(* PLC project SmartTextile_Ladder, Eesha Masand Smart Textile Manufacturing 2 *)
(* stored: creationDateTime 2026-10-07T12:00:00, modificationDateTime 2026-10-07T12:00:00 *)

(* Smart textile line: control logic as a ladder diagram. Runs first in the scan. *)
PROGRAM SmartTextileLadder
  VAR
    X0_StartPB AT %QX102.0 : BOOL;  (* X0: Start push-button (physical) *)
    X1_StopPB AT %QX102.1 : BOOL;  (* X1: Stop push-button (physical) *)
    X2_ResetPB AT %QX102.2 : BOOL;  (* X2: Reset push-button (physical) *)
    X3_AtS1_FeedId AT %QX102.3 : BOOL;  (* X3: Product at station 1: feed / identification *)
    X4_TypeA_Sensor AT %QX102.4 : BOOL;  (* X4: Type A sensor *)
    X5_TypeB_Sensor AT %QX102.5 : BOOL;  (* X5: Type B sensor *)
    X6_AtS2_Cutting AT %QX102.6 : BOOL;  (* X6: Product at station 2: cutting *)
    X7_AtS3_Finishing AT %QX102.7 : BOOL;  (* X7: Product at station 3: finishing *)
    X10_AtS4_Inspection AT %QX103.0 : BOOL;  (* X10: Product at station 4: inspection *)
    X11_InspComplete AT %QX103.1 : BOOL;  (* X11: Inspection complete (vision result valid) *)
    X12_DefectDetected AT %QX103.2 : BOOL;  (* X12: Defect detected by vision *)
    X13_RobotReady AT %QX103.3 : BOOL;  (* X13: Robot ready (home position) *)
    X14_RobotPlaceDone AT %QX103.4 : BOOL;  (* X14: Robot place done *)
    X15_PackComplete AT %QX103.5 : BOOL;  (* X15: Packaging complete *)
    X16_RobotHealthy AT %QX103.6 : BOOL;  (* X16: Robot healthy (NC wiring: ON = OK, OFF = fault) *)
    X17_EStopOK AT %QX103.7 : BOOL;  (* X17: Emergency stop chain (NC wiring: ON = released, OFF = pressed) *)
    X20_AtS5_Robot AT %QX104.0 : BOOL;  (* X20: Product at station 5: robot pick *)
    Y0_FeederMotor AT %QX0.0 : BOOL;  (* Y0: Feeder motor *)
    Y1_MainConveyor AT %QX0.1 : BOOL;  (* Y1: Main conveyor *)
    Y2_Cutter AT %QX0.2 : BOOL;  (* Y2: Cutter (stage 1) *)
    Y3_HeatPress AT %QX0.3 : BOOL;  (* Y3: Heat press (stage 2) *)
    Y4_InspTrigger AT %QX0.4 : BOOL;  (* Y4: Inspection trigger (camera) *)
    Y5_RobotPickReq AT %QX0.5 : BOOL;  (* Y5: Robot pick request *)
    Y6_DestGood AT %QX0.6 : BOOL;  (* Y6: Robot destination: good *)
    Y7_DestReject AT %QX0.7 : BOOL;  (* Y7: Robot destination: reject *)
    Y10_PackMachine AT %QX1.0 : BOOL;  (* Y10: Packaging machine *)
    Y11_AlarmBuzzer AT %QX1.1 : BOOL;  (* Y11: Alarm buzzer *)
    Y12_RunLamp AT %QX1.2 : BOOL;  (* Y12: Run lamp (green) *)
    Y13_FaultLamp AT %QX1.3 : BOOL;  (* Y13: Fault / E-stop lamp (red) *)
    M100_HmiStart AT %QX100.0 : BOOL;  (* M100: HMI start button *)
    M101_HmiStop AT %QX100.1 : BOOL;  (* M101: HMI stop button *)
    M102_HmiReset AT %QX100.2 : BOOL;  (* M102: HMI reset button *)
    M103_HmiAuto AT %QX100.3 : BOOL;  (* M103: HMI auto mode button *)
    M104_HmiManual AT %QX100.4 : BOOL;  (* M104: HMI manual mode button *)
    M105_HmiProdA AT %QX100.5 : BOOL;  (* M105: HMI product A override *)
    M106_HmiProdB AT %QX100.6 : BOOL;  (* M106: HMI product B override *)
    M107_HmiClear AT %QX100.7 : BOOL;  (* M107: HMI clear counters button *)
    M108_HmiEStop AT %QX101.0 : BOOL;  (* M108: HMI emergency stop button *)
    M0_SystemRun AT %QX105.0 : BOOL;  (* M0: System run *)
    M1_Fault AT %QX105.1 : BOOL;  (* M1: Fault latched *)
    M2_EStop AT %QX105.2 : BOOL;  (* M2: Emergency stop latched *)
    M31_ManualMode AT %QX105.3 : BOOL;  (* M31: Manual mode (0 = auto) *)
    M17_ManualTypeB AT %QX105.4 : BOOL;  (* M17: Manual product selection (0 = A, 1 = B) *)
    M3_PhaseIndex AT %QX105.5 : BOOL;  (* M3: Phase: conveyor indexing *)
    M4_PhaseWork AT %QX105.6 : BOOL;  (* M4: Phase: stations working *)
    M75_PackBusy AT %QX105.7 : BOOL;  (* M75: Packaging machine busy *)
    M50_S1_Occupied AT %QX106.0 : BOOL;  (* M50: Station 1 occupied *)
    M51_S2_Occupied AT %QX106.1 : BOOL;  (* M51: Station 2 occupied *)
    M52_S3_Occupied AT %QX106.2 : BOOL;  (* M52: Station 3 occupied *)
    M53_S4_Occupied AT %QX106.3 : BOOL;  (* M53: Station 4 occupied *)
    M54_S5_Occupied AT %QX106.4 : BOOL;  (* M54: Station 5 occupied *)
    M55_DefectAtS4 AT %QX106.5 : BOOL;  (* M55: Defect flag of the product at station 4 *)
    M56_DefectAtS5 AT %QX106.6 : BOOL;  (* M56: Defect flag of the product at station 5 *)
    M60_S1_IsTypeB AT %QX107.0 : BOOL;  (* M60: Product at station 1 is type B *)
    M61_S2_IsTypeB AT %QX107.1 : BOOL;  (* M61: Product at station 2 is type B *)
    M62_S3_IsTypeB AT %QX107.2 : BOOL;  (* M62: Product at station 3 is type B *)
    M63_S4_IsTypeB AT %QX107.3 : BOOL;  (* M63: Product at station 4 is type B *)
    M64_S5_IsTypeB AT %QX107.4 : BOOL;  (* M64: Product at station 5 is type B *)
  END_VAR
  VAR
    M69_FeedDone : BOOL;  (* M69: Feed time elapsed in this work phase *)
    M70_S1_IdDone : BOOL;  (* M70: Station 1 identification done *)
    M71_S2_CutDone : BOOL;  (* M71: Station 2 cutting done *)
    M72_S3_FinishDone : BOOL;  (* M72: Station 3 finishing done *)
    M73_S4_InspDone : BOOL;  (* M73: Station 4 inspection result latched *)
    M80_S1_Departed : BOOL;  (* M80: Old product has left station 1 (this index) *)
    M81_S2_Departed : BOOL;  (* M81: Old product has left station 2 (this index) *)
    M82_S3_Departed : BOOL;  (* M82: Old product has left station 3 (this index) *)
    M83_S4_Departed : BOOL;  (* M83: Old product has left station 4 (this index) *)
    M84_S5_Departed : BOOL;  (* M84: Old product has left station 5 (this index) *)
    M22_GoodSorted : BOOL;  (* M22: Good product sorted (pulse) *)
    M23_RejectSorted : BOOL;  (* M23: Reject product sorted (pulse) *)
    M24_IndexComplete : BOOL;  (* M24: Index complete: all products at next station *)
    M25_WorkComplete : BOOL;  (* M25: Work complete: all stations finished *)
    M26_StationsDone : BOOL;  (* M26: All occupied stations finished their task *)
    M28_AllDeparted : BOOL;  (* M28: Every old product has left its station *)
    M29_AllArrived : BOOL;  (* M29: Every expected product reached its station *)
    M32_PackagedPulse : BOOL;  (* M32: Product packaged (pulse) *)
  END_VAR
  VAR_EXTERNAL
    T0_FeedTime_Q : BOOL;  (* Shared with the data program *)
    T1_CutTime_Q : BOOL;  (* Shared with the data program *)
    T2_FinishA_Q : BOOL;  (* Shared with the data program *)
    T3_FinishB_Q : BOOL;  (* Shared with the data program *)
    T4_InspTimeout_Q : BOOL;  (* Shared with the data program *)
    T7_IndexWdg_Q : BOOL;  (* Shared with the data program *)
    T8_IdDwell_Q : BOOL;  (* Shared with the data program *)
    T9_IdTimeout_Q : BOOL;  (* Shared with the data program *)
    T10_RobotWdg_Q : BOOL;  (* Shared with the data program *)
    T11_PackWdg_Q : BOOL;  (* Shared with the data program *)
    F_R01_RobotFaultRobot : BOOL;  (* Shared with the data program *)
    F_R02_InspectionTimeoutVision : BOOL;  (* Shared with the data program *)
    F_R03_IndexPackagingTimeout : BOOL;  (* Shared with the data program *)
    F_R04_UnknownProductIdentification : BOOL;  (* Shared with the data program *)
    F_R05_EmergencyStopChain : BOOL;  (* Shared with the data program *)
    F_R06_ResetClearFaults : BOOL;  (* Shared with the data program *)
    F_R11_ManualOverrideProduct : BOOL;  (* Shared with the data program *)
    F_R12_ManualOverrideProduct : BOOL;  (* Shared with the data program *)
    F_R13_IdleStartFeed : BOOL;  (* Shared with the data program *)
    F_R26_IndexWork : BOOL;  (* Shared with the data program *)
    F_R27_FeederStartBelt : BOOL;  (* Shared with the data program *)
    F_R29_IdentificationDwell : BOOL;  (* Shared with the data program *)
    F_R30_IdentificationTimeout : BOOL;  (* Shared with the data program *)
    F_R31_IdentifyProductAuto : BOOL;  (* Shared with the data program *)
    F_R32_IdentifyProductB : BOOL;  (* Shared with the data program *)
    F_R35_CutterCuttingTime : BOOL;  (* Shared with the data program *)
    F_R38_FinishingTimeProduct : BOOL;  (* Shared with the data program *)
    F_R39_FinishingTimeProduct : BOOL;  (* Shared with the data program *)
    F_R42_InspectionTimeoutTimer : BOOL;  (* Shared with the data program *)
    F_R49_RobotWatchdogTimer : BOOL;  (* Shared with the data program *)
    F_R54_PackagingMachineWatchdog : BOOL;  (* Shared with the data program *)
    F_R59_WorkIndex : BOOL;  (* Shared with the data program *)
    F_R61_IndexWatchdog15 : BOOL;  (* Shared with the data program *)
    F_R62_StopwatchesAddOne : BOOL;  (* Shared with the data program *)
    F_R63_TaktTimeLast : BOOL;  (* Shared with the data program *)
    F_R64_GoodCounter : BOOL;  (* Shared with the data program *)
    F_R65_RejectCounter : BOOL;  (* Shared with the data program *)
    F_R66_PackagedCounter : BOOL;  (* Shared with the data program *)
    F_R71_ClearCountersKPIs : BOOL;  (* Shared with the data program *)
  END_VAR
  VAR  (* added by the conversion: wires and edge detectors of the diagram *)
    R_TRIG1 : R_TRIG;
    R_TRIG2 : R_TRIG;
    R_TRIG3 : R_TRIG;
    R_TRIG4 : R_TRIG;
    R_TRIG5 : R_TRIG;
    R_TRIG6 : R_TRIG;
    R_TRIG7 : R_TRIG;
    R_TRIG8 : R_TRIG;
  END_VAR

(* LD diagram, written out as Structured Text *)
IF NOT X16_RobotHealthy OR T10_RobotWdg_Q THEN M1_Fault := TRUE; END_IF;
F_R01_RobotFaultRobot := NOT X16_RobotHealthy OR T10_RobotWdg_Q;
IF T4_InspTimeout_Q THEN M1_Fault := TRUE; END_IF;
F_R02_InspectionTimeoutVision := T4_InspTimeout_Q;
IF T7_IndexWdg_Q OR T11_PackWdg_Q THEN M1_Fault := TRUE; END_IF;
F_R03_IndexPackagingTimeout := T7_IndexWdg_Q OR T11_PackWdg_Q;
IF T9_IdTimeout_Q THEN M1_Fault := TRUE; END_IF;
F_R04_UnknownProductIdentification := T9_IdTimeout_Q;
R_TRIG1(CLK := M108_HmiEStop);
F_R05_EmergencyStopChain := NOT X17_EStopOK OR R_TRIG1.Q OR M2_EStop;
IF F_R05_EmergencyStopChain THEN M2_EStop := TRUE; END_IF;
R_TRIG2(CLK := M102_HmiReset);
R_TRIG3(CLK := X2_ResetPB);
F_R06_ResetClearFaults := (R_TRIG2.Q OR R_TRIG3.Q) AND X16_RobotHealthy AND X17_EStopOK;
IF F_R06_ResetClearFaults THEN M1_Fault := FALSE; END_IF;
IF F_R06_ResetClearFaults THEN M2_EStop := FALSE; END_IF;
IF F_R06_ResetClearFaults THEN M3_PhaseIndex := FALSE; END_IF;
IF F_R06_ResetClearFaults THEN M4_PhaseWork := FALSE; END_IF;
IF F_R06_ResetClearFaults THEN M50_S1_Occupied := FALSE; END_IF;
IF F_R06_ResetClearFaults THEN M51_S2_Occupied := FALSE; END_IF;
IF F_R06_ResetClearFaults THEN M52_S3_Occupied := FALSE; END_IF;
IF F_R06_ResetClearFaults THEN M53_S4_Occupied := FALSE; END_IF;
IF F_R06_ResetClearFaults THEN M54_S5_Occupied := FALSE; END_IF;
IF F_R06_ResetClearFaults THEN M55_DefectAtS4 := FALSE; END_IF;
IF F_R06_ResetClearFaults THEN M56_DefectAtS5 := FALSE; END_IF;
IF F_R06_ResetClearFaults THEN M60_S1_IsTypeB := FALSE; END_IF;
IF F_R06_ResetClearFaults THEN M61_S2_IsTypeB := FALSE; END_IF;
IF F_R06_ResetClearFaults THEN M62_S3_IsTypeB := FALSE; END_IF;
IF F_R06_ResetClearFaults THEN M63_S4_IsTypeB := FALSE; END_IF;
IF F_R06_ResetClearFaults THEN M64_S5_IsTypeB := FALSE; END_IF;
IF F_R06_ResetClearFaults THEN M69_FeedDone := FALSE; END_IF;
IF F_R06_ResetClearFaults THEN M70_S1_IdDone := FALSE; END_IF;
IF F_R06_ResetClearFaults THEN M71_S2_CutDone := FALSE; END_IF;
IF F_R06_ResetClearFaults THEN M72_S3_FinishDone := FALSE; END_IF;
IF F_R06_ResetClearFaults THEN M73_S4_InspDone := FALSE; END_IF;
IF F_R06_ResetClearFaults THEN M75_PackBusy := FALSE; END_IF;
IF F_R06_ResetClearFaults THEN M80_S1_Departed := FALSE; END_IF;
IF F_R06_ResetClearFaults THEN M81_S2_Departed := FALSE; END_IF;
IF F_R06_ResetClearFaults THEN M82_S3_Departed := FALSE; END_IF;
IF F_R06_ResetClearFaults THEN M83_S4_Departed := FALSE; END_IF;
IF F_R06_ResetClearFaults THEN M84_S5_Departed := FALSE; END_IF;
R_TRIG4(CLK := M100_HmiStart);
R_TRIG5(CLK := X0_StartPB);
IF (R_TRIG4.Q OR R_TRIG5.Q) AND NOT M1_Fault AND NOT M2_EStop AND X16_RobotHealthy AND X17_EStopOK THEN M0_SystemRun := TRUE; END_IF;
IF M101_HmiStop OR X1_StopPB OR NOT X16_RobotHealthy OR NOT X17_EStopOK OR M1_Fault OR M2_EStop THEN M0_SystemRun := FALSE; END_IF;
IF M103_HmiAuto THEN M31_ManualMode := FALSE; END_IF;
IF M104_HmiManual THEN M31_ManualMode := TRUE; END_IF;
IF M105_HmiProdA AND M31_ManualMode THEN M17_ManualTypeB := FALSE; END_IF;
F_R11_ManualOverrideProduct := M105_HmiProdA AND M31_ManualMode;
IF M106_HmiProdB AND M31_ManualMode THEN M17_ManualTypeB := TRUE; END_IF;
F_R12_ManualOverrideProduct := M106_HmiProdB AND M31_ManualMode;
F_R13_IdleStartFeed := M0_SystemRun AND NOT M3_PhaseIndex AND NOT M4_PhaseWork AND NOT M1_Fault AND NOT M2_EStop;
IF F_R13_IdleStartFeed THEN M4_PhaseWork := TRUE; END_IF;
M28_AllDeparted := M0_SystemRun AND M3_PhaseIndex AND (NOT M50_S1_Occupied OR M80_S1_Departed) AND (NOT M51_S2_Occupied OR M81_S2_Departed) AND (NOT M52_S3_Occupied OR M82_S3_Departed) AND (NOT M53_S4_Occupied OR M83_S4_Departed) AND (NOT M54_S5_Occupied OR M84_S5_Departed);
M29_AllArrived := M0_SystemRun AND M3_PhaseIndex AND X3_AtS1_FeedId AND (NOT M50_S1_Occupied OR X6_AtS2_Cutting) AND (NOT M51_S2_Occupied OR X7_AtS3_Finishing) AND (NOT M52_S3_Occupied OR X10_AtS4_Inspection) AND (NOT M53_S4_Occupied OR X20_AtS5_Robot);
M24_IndexComplete := M28_AllDeparted AND M29_AllArrived;
IF M0_SystemRun AND M3_PhaseIndex AND M50_S1_Occupied AND NOT X3_AtS1_FeedId THEN M80_S1_Departed := TRUE; END_IF;
IF M0_SystemRun AND M3_PhaseIndex AND M51_S2_Occupied AND NOT X6_AtS2_Cutting THEN M81_S2_Departed := TRUE; END_IF;
IF M0_SystemRun AND M3_PhaseIndex AND M52_S3_Occupied AND NOT X7_AtS3_Finishing THEN M82_S3_Departed := TRUE; END_IF;
IF M0_SystemRun AND M3_PhaseIndex AND M53_S4_Occupied AND NOT X10_AtS4_Inspection THEN M83_S4_Departed := TRUE; END_IF;
IF M0_SystemRun AND M3_PhaseIndex AND M54_S5_Occupied AND NOT X20_AtS5_Robot THEN M84_S5_Departed := TRUE; END_IF;
IF M24_IndexComplete AND M53_S4_Occupied THEN M54_S5_Occupied := TRUE; END_IF;
IF M24_IndexComplete AND NOT M53_S4_Occupied THEN M54_S5_Occupied := FALSE; END_IF;
IF M24_IndexComplete AND M52_S3_Occupied THEN M53_S4_Occupied := TRUE; END_IF;
IF M24_IndexComplete AND NOT M52_S3_Occupied THEN M53_S4_Occupied := FALSE; END_IF;
IF M24_IndexComplete AND M51_S2_Occupied THEN M52_S3_Occupied := TRUE; END_IF;
IF M24_IndexComplete AND NOT M51_S2_Occupied THEN M52_S3_Occupied := FALSE; END_IF;
IF M24_IndexComplete AND M50_S1_Occupied THEN M51_S2_Occupied := TRUE; END_IF;
IF M24_IndexComplete AND NOT M50_S1_Occupied THEN M51_S2_Occupied := FALSE; END_IF;
IF M24_IndexComplete THEN M50_S1_Occupied := TRUE; END_IF;
IF M24_IndexComplete AND M63_S4_IsTypeB THEN M64_S5_IsTypeB := TRUE; END_IF;
IF M24_IndexComplete AND NOT M63_S4_IsTypeB THEN M64_S5_IsTypeB := FALSE; END_IF;
IF M24_IndexComplete AND M62_S3_IsTypeB THEN M63_S4_IsTypeB := TRUE; END_IF;
IF M24_IndexComplete AND NOT M62_S3_IsTypeB THEN M63_S4_IsTypeB := FALSE; END_IF;
IF M24_IndexComplete AND M61_S2_IsTypeB THEN M62_S3_IsTypeB := TRUE; END_IF;
IF M24_IndexComplete AND NOT M61_S2_IsTypeB THEN M62_S3_IsTypeB := FALSE; END_IF;
IF M24_IndexComplete AND M60_S1_IsTypeB THEN M61_S2_IsTypeB := TRUE; END_IF;
IF M24_IndexComplete AND NOT M60_S1_IsTypeB THEN M61_S2_IsTypeB := FALSE; END_IF;
IF M24_IndexComplete THEN M60_S1_IsTypeB := FALSE; END_IF;
IF M24_IndexComplete AND M55_DefectAtS4 THEN M56_DefectAtS5 := TRUE; END_IF;
IF M24_IndexComplete AND NOT M55_DefectAtS4 THEN M56_DefectAtS5 := FALSE; END_IF;
IF M24_IndexComplete THEN M55_DefectAtS4 := FALSE; END_IF;
IF M24_IndexComplete THEN M69_FeedDone := FALSE; END_IF;
IF M24_IndexComplete THEN M70_S1_IdDone := FALSE; END_IF;
IF M24_IndexComplete THEN M71_S2_CutDone := FALSE; END_IF;
IF M24_IndexComplete THEN M72_S3_FinishDone := FALSE; END_IF;
IF M24_IndexComplete THEN M73_S4_InspDone := FALSE; END_IF;
IF M24_IndexComplete THEN M80_S1_Departed := FALSE; END_IF;
IF M24_IndexComplete THEN M81_S2_Departed := FALSE; END_IF;
IF M24_IndexComplete THEN M82_S3_Departed := FALSE; END_IF;
IF M24_IndexComplete THEN M83_S4_Departed := FALSE; END_IF;
IF M24_IndexComplete THEN M84_S5_Departed := FALSE; END_IF;
IF M24_IndexComplete THEN M3_PhaseIndex := FALSE; END_IF;
IF M24_IndexComplete THEN M4_PhaseWork := TRUE; END_IF;
F_R26_IndexWork := M24_IndexComplete;
Y0_FeederMotor := M0_SystemRun AND M4_PhaseWork AND NOT M69_FeedDone;
F_R27_FeederStartBelt := M0_SystemRun AND M4_PhaseWork AND NOT M69_FeedDone;
IF T0_FeedTime_Q THEN M69_FeedDone := TRUE; END_IF;
F_R29_IdentificationDwell := M0_SystemRun AND M4_PhaseWork AND M50_S1_Occupied AND X3_AtS1_FeedId;
F_R30_IdentificationTimeout := M0_SystemRun AND M4_PhaseWork AND M50_S1_Occupied AND X3_AtS1_FeedId AND NOT M70_S1_IdDone;
IF T8_IdDwell_Q AND NOT M31_ManualMode AND X4_TypeA_Sensor AND NOT X5_TypeB_Sensor THEN M60_S1_IsTypeB := FALSE; END_IF;
F_R31_IdentifyProductAuto := T8_IdDwell_Q AND NOT M31_ManualMode AND X4_TypeA_Sensor AND NOT X5_TypeB_Sensor;
IF T8_IdDwell_Q AND NOT M31_ManualMode AND X5_TypeB_Sensor AND NOT X4_TypeA_Sensor THEN M60_S1_IsTypeB := TRUE; END_IF;
F_R32_IdentifyProductB := T8_IdDwell_Q AND NOT M31_ManualMode AND X5_TypeB_Sensor AND NOT X4_TypeA_Sensor;
IF T8_IdDwell_Q AND M31_ManualMode AND M17_ManualTypeB THEN M60_S1_IsTypeB := TRUE; END_IF;
IF T8_IdDwell_Q AND M31_ManualMode AND NOT M17_ManualTypeB THEN M60_S1_IsTypeB := FALSE; END_IF;
IF T8_IdDwell_Q AND (M31_ManualMode OR X4_TypeA_Sensor AND NOT X5_TypeB_Sensor OR NOT X4_TypeA_Sensor AND X5_TypeB_Sensor) THEN M70_S1_IdDone := TRUE; END_IF;
Y2_Cutter := M0_SystemRun AND M4_PhaseWork AND M51_S2_Occupied AND X6_AtS2_Cutting AND NOT M71_S2_CutDone;
F_R35_CutterCuttingTime := M0_SystemRun AND M4_PhaseWork AND M51_S2_Occupied AND X6_AtS2_Cutting AND NOT M71_S2_CutDone;
IF T1_CutTime_Q THEN M71_S2_CutDone := TRUE; END_IF;
Y3_HeatPress := M0_SystemRun AND M4_PhaseWork AND M52_S3_Occupied AND X7_AtS3_Finishing AND NOT M72_S3_FinishDone;
F_R38_FinishingTimeProduct := M0_SystemRun AND M4_PhaseWork AND M52_S3_Occupied AND X7_AtS3_Finishing AND NOT M72_S3_FinishDone AND NOT M62_S3_IsTypeB;
F_R39_FinishingTimeProduct := M0_SystemRun AND M4_PhaseWork AND M52_S3_Occupied AND X7_AtS3_Finishing AND NOT M72_S3_FinishDone AND M62_S3_IsTypeB;
IF T2_FinishA_Q OR T3_FinishB_Q THEN M72_S3_FinishDone := TRUE; END_IF;
Y4_InspTrigger := M0_SystemRun AND M4_PhaseWork AND M53_S4_Occupied AND X10_AtS4_Inspection AND NOT M73_S4_InspDone;
F_R42_InspectionTimeoutTimer := M0_SystemRun AND M4_PhaseWork AND M53_S4_Occupied AND X10_AtS4_Inspection AND NOT M73_S4_InspDone AND NOT X11_InspComplete;
IF M0_SystemRun AND M4_PhaseWork AND M53_S4_Occupied AND X10_AtS4_Inspection AND X11_InspComplete AND NOT X12_DefectDetected THEN M55_DefectAtS4 := FALSE; END_IF;
IF M0_SystemRun AND M4_PhaseWork AND M53_S4_Occupied AND X10_AtS4_Inspection AND X11_InspComplete AND X12_DefectDetected THEN M55_DefectAtS4 := TRUE; END_IF;
IF M0_SystemRun AND M4_PhaseWork AND M53_S4_Occupied AND X10_AtS4_Inspection AND X11_InspComplete THEN M73_S4_InspDone := TRUE; END_IF;
Y5_RobotPickReq := M0_SystemRun AND M4_PhaseWork AND M54_S5_Occupied AND X20_AtS5_Robot AND NOT X14_RobotPlaceDone AND (M56_DefectAtS5 OR NOT M75_PackBusy);
Y6_DestGood := M0_SystemRun AND M4_PhaseWork AND M54_S5_Occupied AND NOT M56_DefectAtS5;
Y7_DestReject := M0_SystemRun AND M4_PhaseWork AND M54_S5_Occupied AND M56_DefectAtS5;
F_R49_RobotWatchdogTimer := M0_SystemRun AND M4_PhaseWork AND M54_S5_Occupied;
R_TRIG6(CLK := X14_RobotPlaceDone);
M22_GoodSorted := M0_SystemRun AND M4_PhaseWork AND M54_S5_Occupied AND NOT M56_DefectAtS5 AND R_TRIG6.Q;
R_TRIG7(CLK := X14_RobotPlaceDone);
M23_RejectSorted := M0_SystemRun AND M4_PhaseWork AND M54_S5_Occupied AND M56_DefectAtS5 AND R_TRIG7.Q;
IF M22_GoodSorted OR M23_RejectSorted THEN M54_S5_Occupied := FALSE; END_IF;
IF M22_GoodSorted THEN M75_PackBusy := TRUE; END_IF;
Y10_PackMachine := M0_SystemRun AND M75_PackBusy;
F_R54_PackagingMachineWatchdog := M0_SystemRun AND M75_PackBusy;
R_TRIG8(CLK := X15_PackComplete);
M32_PackagedPulse := M0_SystemRun AND M75_PackBusy AND R_TRIG8.Q;
IF M32_PackagedPulse THEN M75_PackBusy := FALSE; END_IF;
M26_StationsDone := (NOT M50_S1_Occupied OR M70_S1_IdDone) AND (NOT M51_S2_Occupied OR M71_S2_CutDone) AND (NOT M52_S3_Occupied OR M72_S3_FinishDone) AND (NOT M53_S4_Occupied OR M73_S4_InspDone) AND NOT M54_S5_Occupied;
M25_WorkComplete := M0_SystemRun AND M4_PhaseWork AND M69_FeedDone AND M26_StationsDone AND X13_RobotReady;
IF M25_WorkComplete THEN M4_PhaseWork := FALSE; END_IF;
IF M25_WorkComplete THEN M3_PhaseIndex := TRUE; END_IF;
F_R59_WorkIndex := M25_WorkComplete;
Y1_MainConveyor := M0_SystemRun AND M3_PhaseIndex AND NOT M24_IndexComplete;
F_R61_IndexWatchdog15 := M0_SystemRun AND M3_PhaseIndex;
F_R62_StopwatchesAddOne := M0_SystemRun AND (M3_PhaseIndex OR M4_PhaseWork);
F_R63_TaktTimeLast := M22_GoodSorted OR M23_RejectSorted;
F_R64_GoodCounter := M22_GoodSorted;
F_R65_RejectCounter := M23_RejectSorted;
F_R66_PackagedCounter := M32_PackagedPulse;
F_R71_ClearCountersKPIs := M107_HmiClear;
Y12_RunLamp := M0_SystemRun;
Y11_AlarmBuzzer := M1_Fault OR M2_EStop;
Y13_FaultLamp := M1_Fault OR M2_EStop;
END_PROGRAM

(* Timers, counters, fault code, phase and KPI maths. Runs second in the scan. *)
PROGRAM SmartTextileData
  VAR
    D100_GoodCount AT %MW0 : INT;  (* D100: Good count *)
    D101_RejectCount AT %MW1 : INT;  (* D101: Reject count *)
    D102_TotalCount AT %MW2 : INT;  (* D102: Total count *)
    D103_DefectPctX100 AT %MW3 : INT;  (* D103: Defect percentage x100 (1670 = 16.70 %) *)
    D104_TaktTime01s AT %MW4 : INT;  (* D104: Takt time: gap between sorted products (0.1 s) *)
    D105_RateX10PerMin AT %MW5 : INT;  (* D105: Production rate (0.1 products / min) *)
    D106_CurrentProduct AT %MW6 : INT;  (* D106: Product at station 1 (1 = A, 2 = B) *)
    D107_Phase AT %MW7 : INT;  (* D107: Phase (0 idle, 10 indexing, 20 working) *)
    D108_FaultCode AT %MW8 : INT;  (* D108: Fault code (0 none, 1-5) *)
    D109_PackagedCount AT %MW9 : INT;  (* D109: Packaged count *)
  END_VAR
  VAR
    D110_CycleMs : DINT;  (* D110: Takt stopwatch (ms, scan based) *)
    D111_RunMs : DINT;  (* D111: Running time stopwatch (ms, scan based) *)
    T0_FeedTime : TON;  (* T0: Feed time 2 s *)
    T1_CutTime : TON;  (* T1: Cutting time 3 s *)
    T2_FinishA : TON;  (* T2: Finishing time, product A 5 s *)
    T3_FinishB : TON;  (* T3: Finishing time, product B 8 s *)
    T4_InspTimeout : TON;  (* T4: Inspection timeout 5 s *)
    T7_IndexWdg : TON;  (* T7: Index watchdog 15 s (jam / no material) *)
    T8_IdDwell : TON;  (* T8: Identification dwell 0.5 s *)
    T9_IdTimeout : TON;  (* T9: Identification timeout 3 s *)
    T10_RobotWdg : TON;  (* T10: Robot watchdog 30 s *)
    T11_PackWdg : TON;  (* T11: Packaging watchdog 15 s *)
    C0_GoodCtr : CTU;  (* C0: Good counter *)
    C1_RejectCtr : CTU;  (* C1: Reject counter *)
    C2_PackagedCtr : CTU;  (* C2: Packaged counter *)
    pw : BOOL;  (* Power flow of the current rung *)
  END_VAR
  VAR_EXTERNAL
    T0_FeedTime_Q : BOOL;  (* Shared with the data program *)
    T1_CutTime_Q : BOOL;  (* Shared with the data program *)
    T2_FinishA_Q : BOOL;  (* Shared with the data program *)
    T3_FinishB_Q : BOOL;  (* Shared with the data program *)
    T4_InspTimeout_Q : BOOL;  (* Shared with the data program *)
    T7_IndexWdg_Q : BOOL;  (* Shared with the data program *)
    T8_IdDwell_Q : BOOL;  (* Shared with the data program *)
    T9_IdTimeout_Q : BOOL;  (* Shared with the data program *)
    T10_RobotWdg_Q : BOOL;  (* Shared with the data program *)
    T11_PackWdg_Q : BOOL;  (* Shared with the data program *)
    F_R01_RobotFaultRobot : BOOL;  (* Shared with the data program *)
    F_R02_InspectionTimeoutVision : BOOL;  (* Shared with the data program *)
    F_R03_IndexPackagingTimeout : BOOL;  (* Shared with the data program *)
    F_R04_UnknownProductIdentification : BOOL;  (* Shared with the data program *)
    F_R05_EmergencyStopChain : BOOL;  (* Shared with the data program *)
    F_R06_ResetClearFaults : BOOL;  (* Shared with the data program *)
    F_R11_ManualOverrideProduct : BOOL;  (* Shared with the data program *)
    F_R12_ManualOverrideProduct : BOOL;  (* Shared with the data program *)
    F_R13_IdleStartFeed : BOOL;  (* Shared with the data program *)
    F_R26_IndexWork : BOOL;  (* Shared with the data program *)
    F_R27_FeederStartBelt : BOOL;  (* Shared with the data program *)
    F_R29_IdentificationDwell : BOOL;  (* Shared with the data program *)
    F_R30_IdentificationTimeout : BOOL;  (* Shared with the data program *)
    F_R31_IdentifyProductAuto : BOOL;  (* Shared with the data program *)
    F_R32_IdentifyProductB : BOOL;  (* Shared with the data program *)
    F_R35_CutterCuttingTime : BOOL;  (* Shared with the data program *)
    F_R38_FinishingTimeProduct : BOOL;  (* Shared with the data program *)
    F_R39_FinishingTimeProduct : BOOL;  (* Shared with the data program *)
    F_R42_InspectionTimeoutTimer : BOOL;  (* Shared with the data program *)
    F_R49_RobotWatchdogTimer : BOOL;  (* Shared with the data program *)
    F_R54_PackagingMachineWatchdog : BOOL;  (* Shared with the data program *)
    F_R59_WorkIndex : BOOL;  (* Shared with the data program *)
    F_R61_IndexWatchdog15 : BOOL;  (* Shared with the data program *)
    F_R62_StopwatchesAddOne : BOOL;  (* Shared with the data program *)
    F_R63_TaktTimeLast : BOOL;  (* Shared with the data program *)
    F_R64_GoodCounter : BOOL;  (* Shared with the data program *)
    F_R65_RejectCounter : BOOL;  (* Shared with the data program *)
    F_R66_PackagedCounter : BOOL;  (* Shared with the data program *)
    F_R71_ClearCountersKPIs : BOOL;  (* Shared with the data program *)
  END_VAR

            
  (* Timers, counters, fault code, phase, takt time and KPI maths of the line.
     The ladder program SmartTextileLadder runs first in every scan and sets the F_R.. flags,
     this program reads them, runs the timers and counters, and gives back the T.._Q done bits. *)

  (* R1: Robot fault or robot timeout *)
  IF F_R01_RobotFaultRobot THEN D108_FaultCode := 2; END_IF;

  (* R2: Inspection timeout (no vision result) *)
  IF F_R02_InspectionTimeoutVision THEN D108_FaultCode := 1; END_IF;

  (* R3: Index or packaging timeout (jam, no material) *)
  IF F_R03_IndexPackagingTimeout THEN D108_FaultCode := 3; END_IF;

  (* R4: Unknown product (identification failed) *)
  IF F_R04_UnknownProductIdentification THEN D108_FaultCode := 4; END_IF;

  (* R5: Emergency stop (chain open or HMI button) *)
  IF F_R05_EmergencyStopChain THEN D108_FaultCode := 5; END_IF;

  (* R6: Reset: clear faults, E-stop and the line *)
  IF F_R06_ResetClearFaults THEN D107_Phase := 0; END_IF;
  IF F_R06_ResetClearFaults THEN D108_FaultCode := 0; END_IF;
  IF F_R06_ResetClearFaults THEN D110_CycleMs := 0; END_IF;

  (* R11: Manual override: product A *)
  IF F_R11_ManualOverrideProduct THEN D106_CurrentProduct := 1; END_IF;

  (* R12: Manual override: product B *)
  IF F_R12_ManualOverrideProduct THEN D106_CurrentProduct := 2; END_IF;

  (* R13: Idle start: feed the first product *)
  IF F_R13_IdleStartFeed THEN D107_Phase := 20; END_IF;

  (* R26: Index to work *)
  IF F_R26_IndexWork THEN D107_Phase := 20; END_IF;

  (* R27: Feeder at the start of the belt *)
  T0_FeedTime(IN := F_R27_FeederStartBelt, PT := T#2000ms);
  T0_FeedTime_Q := T0_FeedTime.Q;

  (* R29: Identification dwell *)
  T8_IdDwell(IN := F_R29_IdentificationDwell, PT := T#500ms);
  T8_IdDwell_Q := T8_IdDwell.Q;

  (* R30: Identification timeout *)
  T9_IdTimeout(IN := F_R30_IdentificationTimeout, PT := T#3000ms);
  T9_IdTimeout_Q := T9_IdTimeout.Q;

  (* R31: Identify product A (auto mode) *)
  IF F_R31_IdentifyProductAuto THEN D106_CurrentProduct := 1; END_IF;

  (* R32: Identify product B (auto mode) *)
  IF F_R32_IdentifyProductB THEN D106_CurrentProduct := 2; END_IF;

  (* R35: Cutter and cutting time *)
  T1_CutTime(IN := F_R35_CutterCuttingTime, PT := T#3000ms);
  T1_CutTime_Q := T1_CutTime.Q;

  (* R38: Finishing time, product A (5 s) *)
  T2_FinishA(IN := F_R38_FinishingTimeProduct, PT := T#5000ms);
  T2_FinishA_Q := T2_FinishA.Q;

  (* R39: Finishing time, product B (8 s) *)
  T3_FinishB(IN := F_R39_FinishingTimeProduct, PT := T#8000ms);
  T3_FinishB_Q := T3_FinishB.Q;

  (* R42: Inspection timeout timer *)
  T4_InspTimeout(IN := F_R42_InspectionTimeoutTimer, PT := T#5000ms);
  T4_InspTimeout_Q := T4_InspTimeout.Q;

  (* R49: Robot watchdog timer *)
  T10_RobotWdg(IN := F_R49_RobotWatchdogTimer, PT := T#30000ms);
  T10_RobotWdg_Q := T10_RobotWdg.Q;

  (* R54: Packaging machine and watchdog *)
  T11_PackWdg(IN := F_R54_PackagingMachineWatchdog, PT := T#15000ms);
  T11_PackWdg_Q := T11_PackWdg.Q;

  (* R59: Work to index *)
  IF F_R59_WorkIndex THEN D107_Phase := 10; END_IF;

  (* R61: Index watchdog (15 s) *)
  T7_IndexWdg(IN := F_R61_IndexWatchdog15, PT := T#15000ms);
  T7_IndexWdg_Q := T7_IndexWdg.Q;

  (* R62: Stopwatches (add one scan = 20 ms) *)
  IF F_R62_StopwatchesAddOne THEN D110_CycleMs := (D110_CycleMs + 20); END_IF;
  IF F_R62_StopwatchesAddOne THEN D111_RunMs := (D111_RunMs + 20); END_IF;

  (* R63: Takt time of the last product (0.1 s) *)
  IF F_R63_TaktTimeLast THEN D104_TaktTime01s := DINT_TO_INT((D110_CycleMs / 100)); END_IF;
  IF F_R63_TaktTimeLast THEN D110_CycleMs := 0; END_IF;

  (* R64: Good counter *)
  C0_GoodCtr(CU := F_R64_GoodCounter, R := F_R71_ClearCountersKPIs, PV := 9999);

  (* R65: Reject counter *)
  C1_RejectCtr(CU := F_R65_RejectCounter, R := F_R71_ClearCountersKPIs, PV := 9999);

  (* R66: Packaged counter *)
  C2_PackagedCtr(CU := F_R66_PackagedCounter, R := F_R71_ClearCountersKPIs, PV := 9999);

  (* R67: Copy counters to data registers *)
  pw := TRUE;
  IF pw THEN D100_GoodCount := C0_GoodCtr.CV; END_IF;
  IF pw THEN D101_RejectCount := C1_RejectCtr.CV; END_IF;
  IF pw THEN D109_PackagedCount := C2_PackagedCtr.CV; END_IF;

  (* R68: Total count *)
  pw := TRUE;
  IF pw THEN D102_TotalCount := DINT_TO_INT((INT_TO_DINT(D100_GoodCount) + INT_TO_DINT(D101_RejectCount))); END_IF;

  (* R69: Defect percentage x100 *)
  pw := (D102_TotalCount > 0);
  IF pw THEN D103_DefectPctX100 := DINT_TO_INT(((INT_TO_DINT(D101_RejectCount) * 10000) / INT_TO_DINT(D102_TotalCount))); END_IF;

  (* R70: Production rate: average products per minute x10 *)
  pw := (D111_RunMs >= 100);
  IF pw THEN D105_RateX10PerMin := DINT_TO_INT(((INT_TO_DINT(D102_TotalCount) * 6000) / (D111_RunMs / 100))); END_IF;

  (* R71: Clear counters and KPIs (HMI) *)
  IF F_R71_ClearCountersKPIs THEN D103_DefectPctX100 := 0; END_IF;
  IF F_R71_ClearCountersKPIs THEN D104_TaktTime01s := 0; END_IF;
  IF F_R71_ClearCountersKPIs THEN D105_RateX10PerMin := 0; END_IF;
  IF F_R71_ClearCountersKPIs THEN D110_CycleMs := 0; END_IF;
  IF F_R71_ClearCountersKPIs THEN D111_RunMs := 0; END_IF;


          
END_PROGRAM

CONFIGURATION Config0
  VAR_GLOBAL
    T0_FeedTime_Q : BOOL;  (* Shared with the data program *)
    T1_CutTime_Q : BOOL;  (* Shared with the data program *)
    T2_FinishA_Q : BOOL;  (* Shared with the data program *)
    T3_FinishB_Q : BOOL;  (* Shared with the data program *)
    T4_InspTimeout_Q : BOOL;  (* Shared with the data program *)
    T7_IndexWdg_Q : BOOL;  (* Shared with the data program *)
    T8_IdDwell_Q : BOOL;  (* Shared with the data program *)
    T9_IdTimeout_Q : BOOL;  (* Shared with the data program *)
    T10_RobotWdg_Q : BOOL;  (* Shared with the data program *)
    T11_PackWdg_Q : BOOL;  (* Shared with the data program *)
    F_R01_RobotFaultRobot : BOOL;  (* Shared with the data program *)
    F_R02_InspectionTimeoutVision : BOOL;  (* Shared with the data program *)
    F_R03_IndexPackagingTimeout : BOOL;  (* Shared with the data program *)
    F_R04_UnknownProductIdentification : BOOL;  (* Shared with the data program *)
    F_R05_EmergencyStopChain : BOOL;  (* Shared with the data program *)
    F_R06_ResetClearFaults : BOOL;  (* Shared with the data program *)
    F_R11_ManualOverrideProduct : BOOL;  (* Shared with the data program *)
    F_R12_ManualOverrideProduct : BOOL;  (* Shared with the data program *)
    F_R13_IdleStartFeed : BOOL;  (* Shared with the data program *)
    F_R26_IndexWork : BOOL;  (* Shared with the data program *)
    F_R27_FeederStartBelt : BOOL;  (* Shared with the data program *)
    F_R29_IdentificationDwell : BOOL;  (* Shared with the data program *)
    F_R30_IdentificationTimeout : BOOL;  (* Shared with the data program *)
    F_R31_IdentifyProductAuto : BOOL;  (* Shared with the data program *)
    F_R32_IdentifyProductB : BOOL;  (* Shared with the data program *)
    F_R35_CutterCuttingTime : BOOL;  (* Shared with the data program *)
    F_R38_FinishingTimeProduct : BOOL;  (* Shared with the data program *)
    F_R39_FinishingTimeProduct : BOOL;  (* Shared with the data program *)
    F_R42_InspectionTimeoutTimer : BOOL;  (* Shared with the data program *)
    F_R49_RobotWatchdogTimer : BOOL;  (* Shared with the data program *)
    F_R54_PackagingMachineWatchdog : BOOL;  (* Shared with the data program *)
    F_R59_WorkIndex : BOOL;  (* Shared with the data program *)
    F_R61_IndexWatchdog15 : BOOL;  (* Shared with the data program *)
    F_R62_StopwatchesAddOne : BOOL;  (* Shared with the data program *)
    F_R63_TaktTimeLast : BOOL;  (* Shared with the data program *)
    F_R64_GoodCounter : BOOL;  (* Shared with the data program *)
    F_R65_RejectCounter : BOOL;  (* Shared with the data program *)
    F_R66_PackagedCounter : BOOL;  (* Shared with the data program *)
    F_R71_ClearCountersKPIs : BOOL;  (* Shared with the data program *)
  END_VAR
  RESOURCE Res0 ON PLC
    TASK TaskMain(INTERVAL := T#20ms, PRIORITY := 0);
    PROGRAM Inst0 WITH TaskMain : SmartTextileLadder;
    PROGRAM Inst1 WITH TaskMain : SmartTextileData;
  END_RESOURCE
END_CONFIGURATION
